VAR_GLOBAL
	{attribute 'OPC.UA.DA' := '1'}
	OPCModule			: ARRAY [0..ModuleCnt] OF DUT_SERVER_MODULE_INTERFACE;
	{attribute 'OPC.UA.DA' := '1'}
	ProductionList		: ARRAY [0..TaskCnt] OF DUT_SERVER_TASK;
	{attribute 'OPC.UA.DA' := '1'}
	RecipeOffer			: ARRAY [0..OfferCnt] OF DUT_RECIPEOFFER;
	{attribute 'OPC.UA.DA' := '1'}
	RecipeOrder			: ARRAY [0..OrderCnt] OF DUT_RECIPEORDER;
END_VAR

(* stored: Version 1.1.0.1, ProductVersion 3.1.0.25
   GVL GVL: Id {f7c42ae6-b8b3-4b13-9acf-f4bd9d23ea63} *)
